% RSLogix 500 project JSR AND RETURN 1.RSS, saved by version 8.30.00.15 %
PROJECT "UNTITLED"    % processor: MicroLogix 1000 %

PROGRAM FILES
  LAD 2 "MAIN_PROG"  4 rungs
  LAD 3 "USER_FAULT"  2 rungs
  LAD 4 "HSC_INT"  2 rungs
  LAD 5 "STI_INT"  4 rungs
  LAD 6, 7, 8, 9, 10, 11, 12, 13, 14, 15, 16: only END

DATA FILES
  O0 OUTPUT  1 elements
  I1 INPUT  2 elements
  S2 STATUS  33 elements
  B3 BINARY  32 elements
  T4 TIMER  40 elements
  C5 COUNTER  32 elements
  R6 CONTROL  16 elements
  N7 INTEGER  105 elements

LADDER 2 "MAIN_PROG"
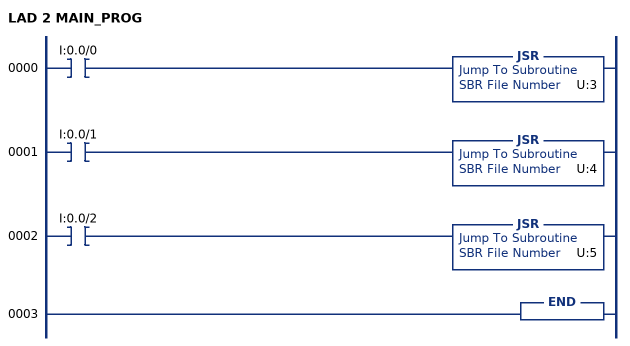
% Rung: 0 %
SOR XIC I:0.0/0 JSR U:3 EOR
% Rung: 1 %
SOR XIC I:0.0/1 JSR U:4 EOR
% Rung: 2 %
SOR XIC I:0.0/2 JSR U:5 EOR
% Rung: 3 %
SOR END EOR

LADDER 3 "USER_FAULT"
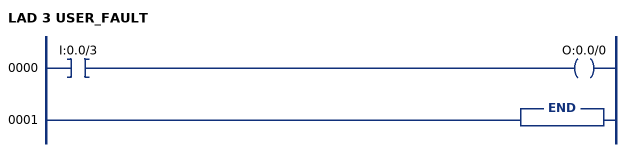
% Rung: 0 %
SOR XIC I:0.0/3 OTE O:0.0/0 EOR
% Rung: 1 %
SOR END EOR

LADDER 4 "HSC_INT"
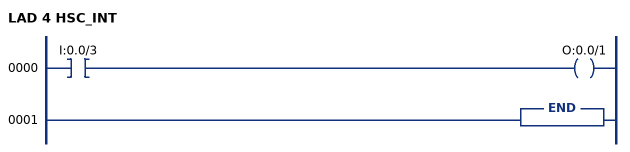
% Rung: 0 %
SOR XIC I:0.0/3 OTE O:0.0/1 EOR
% Rung: 1 %
SOR END EOR

LADDER 5 "STI_INT"
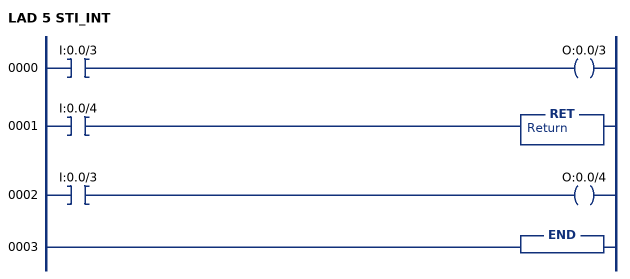
% Rung: 0 %
SOR XIC I:0.0/3 OTE O:0.0/3 EOR
% Rung: 1 %
SOR XIC I:0.0/4 RET EOR
% Rung: 2 %
SOR XIC I:0.0/3 OTE O:0.0/4 EOR
% Rung: 3 %
SOR END EOR
